// TIA Portal V16 export
// export: Created 2024-09-05T17:39:13.0780326Z, ExportSetting WithDefaults, DisplayName Totally Integrated Automation Portal, DisplayVersion V16 Update 6, DisplayName TIA Portal Version Control Interface, DisplayVersion V16 Update 2, DisplayName TIA Portal Openness, DisplayVersion V16 Update 6, DisplayName STEP 7 Professional, DisplayVersion V16 Update 6, DisplayName STEP 7 Safety, DisplayVersion V16, DisplayName WinCC Advanced, DisplayVersion V16 Update 6
FUNCTION "Reader Cognex Dataman" : Void   // FC302, LAD
{ S7_Optimized_Access := 'TRUE' }
VERSION : 0.1
// stored: AutoNumber false, IsIECCheckEnabled false, SetENOAutomatically false, UDAEnableTagReadback false
   VAR_IN_OUT
      ID : "UDT_CognexReaders";
   END_VAR
   VAR_TEMP
      AcquisitionControl : Struct
         TriggerEnable : Bool;
         Trigger : Bool;
         Reserved : Array[2..7] of Bool;
      END_STRUCT;
      AcquisitionStatus : Struct
         TriggerReady : Bool;
         TriggerAck : Bool;
         Reserved : Bool;
         MissedAck : Bool;
         Reserved_1 : Array[4..7] of Bool;
         TriggerID : Word;
      END_STRUCT;
      ResultsControl : Struct
         ResultBufferEnable : Bool;
         ResultsAck : Bool;
         Reserve : Array[2..7] of Bool;
      END_STRUCT;
      ResultsStatus : Struct
         Decoding : Bool;
         "Decode Complete" : Bool;
         "Results Buffer Overrun" : Bool;
         "Results Available" : Bool;
         Reserve_4 : Bool;
         Reserve_5 : Bool;
         Reserve_6 : Bool;
         GeneralFault : Bool;
      END_STRUCT;
      ResultData : Struct
         ID : Word;
         Code : Word;
         Lenght : Word;
         Data : Array[1..64] of Byte;
      END_STRUCT;
      "Return" : Word;
   END_VAR
   VAR_TEMP   // added for the SCL form of the ladder/FBD networks
      _w1 : Bool;
   END_VAR
BEGIN

REGION Network 1: Read input map
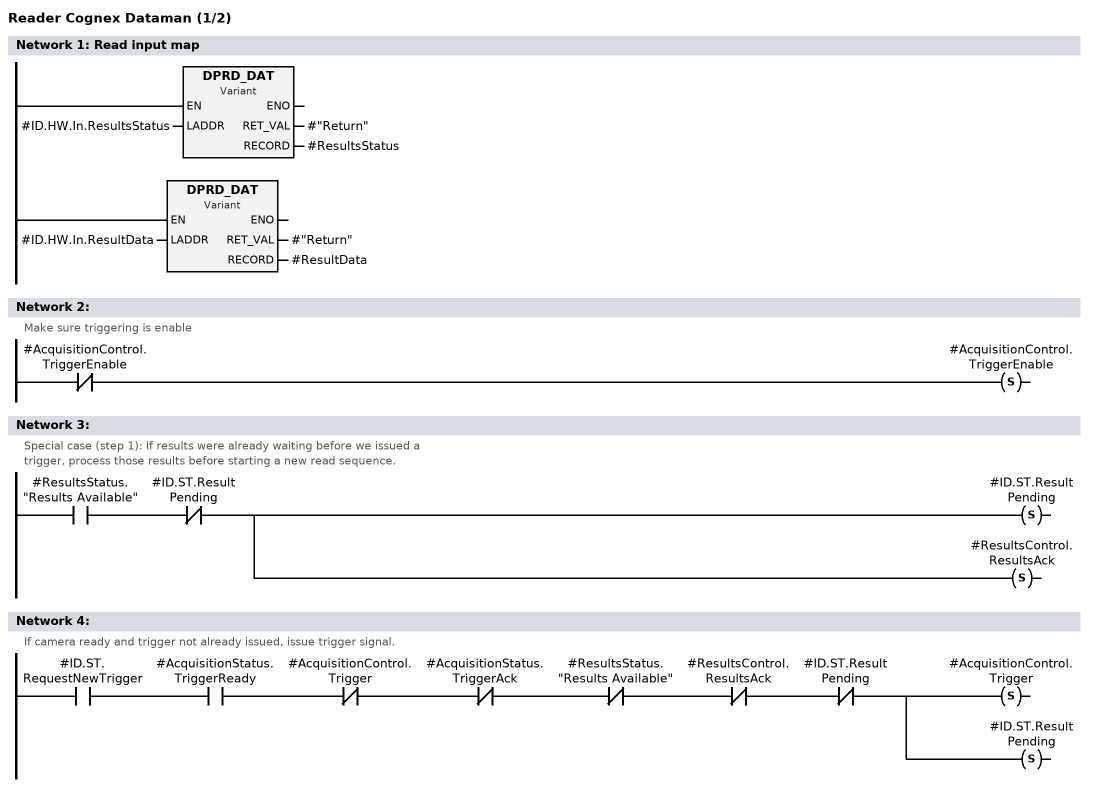
   RUNG wire#powerrail
      { S7_Templates := "[ptr_type := Variant, laddr_type := HW_IO]" } DPRD_DAT(LADDR := #ID.HW.In.ResultsStatus, RET_VAL => #"Return", RECORD => #ResultsStatus)
   END_RUNG
   RUNG wire#powerrail
      { S7_Templates := "[ptr_type := Variant, laddr_type := HW_IO]" } DPRD_DAT(LADDR := #ID.HW.In.ResultData, RET_VAL => #"Return", RECORD => #ResultData)
   END_RUNG
   // the same network as SCL:
   #"Return" := DPRD_DAT(LADDR := #ID.HW.In.ResultsStatus, RECORD => #ResultsStatus);
   #"Return" := DPRD_DAT(LADDR := #ID.HW.In.ResultData, RECORD => #ResultData);
END_REGION

REGION Network 2
   // Make sure triggering is enable
   RUNG wire#powerrail
      I_Contact( #AcquisitionControl.TriggerEnable )
      S_Coil( #AcquisitionControl.TriggerEnable )
   END_RUNG
   // the same network as SCL:
   IF NOT #AcquisitionControl.TriggerEnable THEN #AcquisitionControl.TriggerEnable := TRUE; END_IF;
END_REGION

REGION Network 3
   // Special case (step 1): If results were already waiting before we issued a 
   // trigger, process those results before starting a new read sequence.
   RUNG wire#powerrail
      Contact( #ResultsStatus."Results Available" )
      I_Contact( #ID.ST.ResultPending )
      wire#w1
      S_Coil( #ID.ST.ResultPending )
   END_RUNG
   RUNG wire#w1
      S_Coil( #ResultsControl.ResultsAck )
   END_RUNG
   // the same network as SCL:
   #_w1 := #ResultsStatus."Results Available" AND NOT #ID.ST.ResultPending;
   IF #_w1 THEN
       #ID.ST.ResultPending := TRUE;
       #ResultsControl.ResultsAck := TRUE;
   END_IF;
END_REGION

REGION Network 4
   // If camera ready and trigger not already issued, issue trigger signal.
   RUNG wire#powerrail
      Contact( #ID.ST.RequestNewTrigger )
      Contact( #AcquisitionStatus.TriggerReady )
      I_Contact( #AcquisitionControl.Trigger )
      I_Contact( #AcquisitionStatus.TriggerAck )
      I_Contact( #ResultsStatus."Results Available" )
      I_Contact( #ResultsControl.ResultsAck )
      I_Contact( #ID.ST.ResultPending )
      wire#w1
      S_Coil( #AcquisitionControl.Trigger )
   END_RUNG
   RUNG wire#w1
      S_Coil( #ID.ST.ResultPending )
   END_RUNG
   // the same network as SCL:
   #_w1 := #ID.ST.RequestNewTrigger AND #AcquisitionStatus.TriggerReady AND NOT #AcquisitionControl.Trigger AND NOT #AcquisitionStatus.TriggerAck AND NOT #ResultsStatus."Results Available" AND NOT #ResultsControl.ResultsAck AND NOT #ID.ST.ResultPending;
   IF #_w1 THEN
       #AcquisitionControl.Trigger := TRUE;
       #ID.ST.ResultPending := TRUE;
   END_IF;
END_REGION

REGION Network 5
   // If results available, get the read results
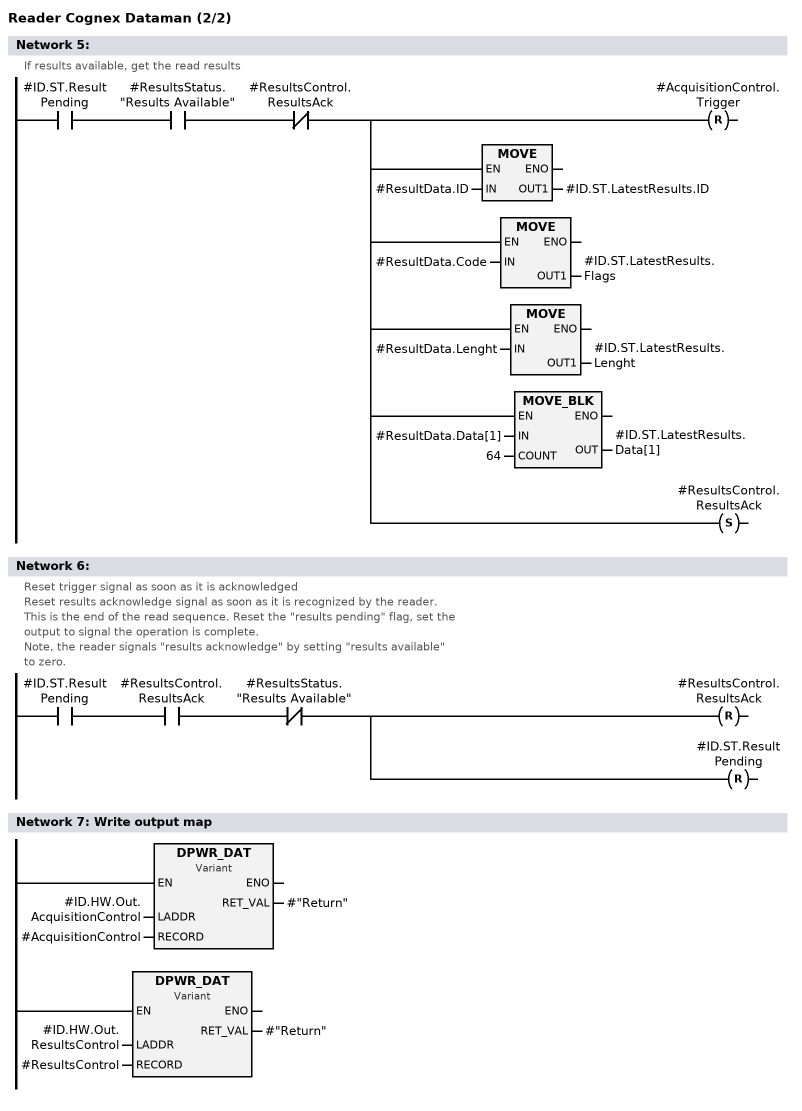
   IF #ID.ST.ResultPending AND #ResultsStatus."Results Available" AND NOT #ResultsControl.ResultsAck THEN
       #AcquisitionControl.Trigger := FALSE;
       #ID.ST.LatestResults.ID := #ResultData.ID;
       #ID.ST.LatestResults.Flags := #ResultData.Code;
       #ID.ST.LatestResults.Lenght := #ResultData.Lenght;
       MOVE_BLK(IN := #ResultData.Data[1], COUNT := 64, OUT => #ID.ST.LatestResults.Data[1]);
       #ResultsControl.ResultsAck := TRUE;
   END_IF;
END_REGION

REGION Network 6
   // Reset trigger signal as soon as it is acknowledged 
   // Reset results acknowledge signal as soon as it is recognized by the reader.
   // 
   // This is the end of the read sequence. Reset the "results pending" flag, set the 
   // output to signal the operation is complete.
   // 
   // Note, the reader signals "results acknowledge" by setting "results available" 
   // to zero.
   RUNG wire#powerrail
      Contact( #ID.ST.ResultPending )
      Contact( #ResultsControl.ResultsAck )
      I_Contact( #ResultsStatus."Results Available" )
      wire#w1
      R_Coil( #ResultsControl.ResultsAck )
   END_RUNG
   RUNG wire#w1
      R_Coil( #ID.ST.ResultPending )
   END_RUNG
   // the same network as SCL:
   #_w1 := #ID.ST.ResultPending AND #ResultsControl.ResultsAck AND NOT #ResultsStatus."Results Available";
   IF #_w1 THEN
       #ResultsControl.ResultsAck := FALSE;
       #ID.ST.ResultPending := FALSE;
   END_IF;
END_REGION

REGION Network 7: Write output map
   RUNG wire#powerrail
      { S7_Templates := "[ptr_type := Variant, laddr_type := HW_IO]" } DPWR_DAT(LADDR := #ID.HW.Out.AcquisitionControl, RECORD := #AcquisitionControl, RET_VAL => #"Return")
   END_RUNG
   RUNG wire#powerrail
      { S7_Templates := "[ptr_type := Variant, laddr_type := HW_IO]" } DPWR_DAT(LADDR := #ID.HW.Out.ResultsControl, RECORD := #ResultsControl, RET_VAL => #"Return")
   END_RUNG
   // the same network as SCL:
   #"Return" := DPWR_DAT(LADDR := #ID.HW.Out.AcquisitionControl, RECORD := #AcquisitionControl);
   #"Return" := DPWR_DAT(LADDR := #ID.HW.Out.ResultsControl, RECORD := #ResultsControl);
END_REGION
END_FUNCTION
